{region '#Template'}
	{attribute 'Version' := '5.2.1.0'}
	{attribute 'Tags' := '"LCID": "1031", "Text": "RA, Sunprotection, Building"'}
	{attribute 'Tags' := '"LCID": "1033", "Text": "RA, Sunprotection, Building"'}
	{attribute 'Using' := '"Type": "Template", "URI": "Site"'}
	{attribute 'Using' := '"Type": "Template", "URI": "BA2_Param"'}
	{attribute 'Using' := '"Type": "Template", "URI": "EC_ID"'}
	{attribute 'Using' := '"Type": "Template", "URI": "ST_BA_BuildingSunblind"'}
	{attribute 'Using' := '"Type": "Template", "URI": "ST_BA_Sunblind"'}
	{attribute 'Using' := '"Type": "Template", "URI": "E_BA_SunBldPrio"'}
	{attribute 'Description' := '"LCID": "1031", "Text": "Sonnenschutz Gebäudedaten"'}
	{attribute 'Description' := '"LCID": "1033", "Text": "Sunprotection building data"'}
{endregion}
FUNCTION_BLOCK FB_BA_BuildingSunprotection EXTENDS FB_BA_View
VAR_INPUT CONSTANT	
	FireAlert					: FB_BA_SunBldEvt			:=(ePrio:=E_BA_SunBldPrio.eFire);	
	Burglary					: FB_BA_SunBldEvt			:=(ePrio:=E_BA_SunBldPrio.eBurglary);	
	IceProtection				: FB_BA_IceProtection;  
	GlobalThAutoRlse			: FB_BA_Hys_03;
	GlobalTwiLgtAutoRlse		: FB_BA_Hys_03;
	SunPrtcPosIntval			: FB_BA_AV_Op_SP;       
	GlobalResetManMode			: FB_BA_BV_Op_Val;   
END_VAR

VAR
	BuildingAlarms				: FB_BA_SunBldTgmSel4;	
	rtManResetEnergLvl			: R_TRIG;	
END_VAR
VAR // added by the converter: edge detectors and wires of the graphical bodies
    _s1 : ST_BA_BuildingSunblind;
    _w1 : UDINT;
END_VAR

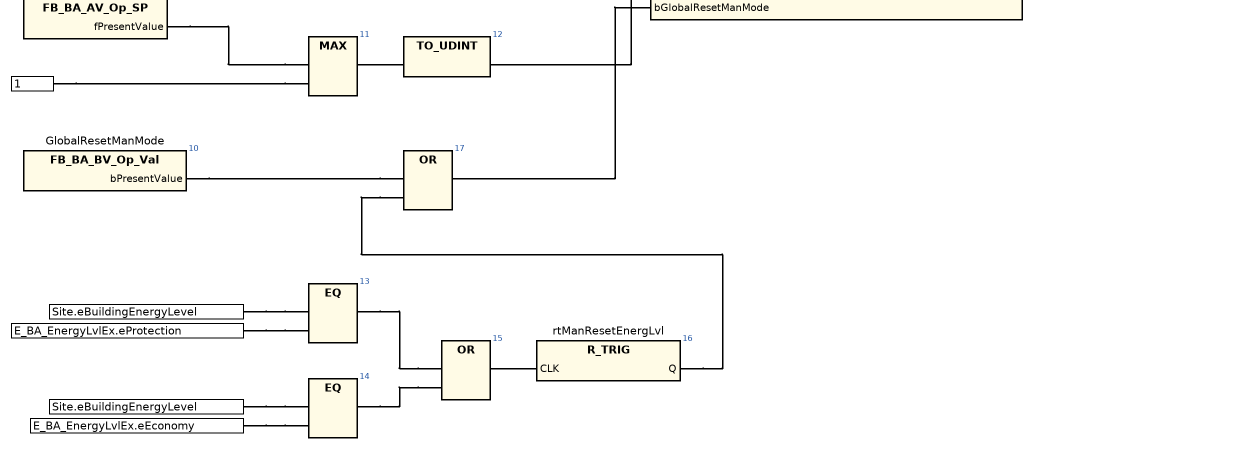
SUPER^(); // FB_BA_View
IceProtection(); // FB_BA_IceProtection
// ----------------------------------------  common alarms  ----------------------------------------
FireAlert(bEn := Site.stBuildingAlarms.bFireAlert, fPos := 0.0, fAngl := 0.0); // FB_BA_SunBldEvt
Burglary(bEn := Site.stBuildingAlarms.bBurglary, fPos := 0.0, fAngl := 0.0); // FB_BA_SunBldEvt
BuildingAlarms(
    stSunBldTgm_1 := FireAlert.stSunBld,
    stSunBldTgm_2 := Burglary.stSunBld,
    stSunBldTgm_3 := IceProtection.stSunBld); // FB_BA_SunBldTgmSel4
// ----------------------------------------  global criteria thermo- and twilight-automatic  ----------------------------------------
GlobalThAutoRlse(bEn := TRUE, fIn := Site.stWeatherStation.fGlobalRadiation); // FB_BA_Hys_03
GlobalTwiLgtAutoRlse(bEn := TRUE, fIn := (Site.stWeatherStation.fBrightnessNorth + Site.stWeatherStation.fBrightnessEast + Site.stWeatherStation.fBrightnessSouth + Site.stWeatherStation.fBrightnessWest) / 4); // FB_BA_Hys_03
// ----------------------------------------  assembling building-data-telegram  ----------------------------------------
SunPrtcPosIntval(); // FB_BA_AV_Op_SP
GlobalResetManMode(); // FB_BA_BV_Op_Val
_w1 := TO_UDINT(MAX(SunPrtcPosIntval.fPresentValue, 1));
rtManResetEnergLvl(CLK := Site.eBuildingEnergyLevel = E_BA_EnergyLvlEx.eProtection OR Site.eBuildingEnergyLevel = E_BA_EnergyLvlEx.eEconomy); // R_TRIG
// compose _s1 : ST_BA_BuildingSunblind
_s1.stSunBld := BuildingAlarms.stSunBld;
_s1.bGlobalThAuto_Release := GlobalThAutoRlse.bPresentValue;
_s1.bGlobalTwiLgtAuto_Release := GlobalTwiLgtAutoRlse.bPresentValue;
_s1.nSunPrtc_PositionInterval := _w1;
_s1.bGlobalResetManMode := GlobalResetManMode.bPresentValue OR rtManResetEnergLvl.Q;
Site.stBuildingSunBlind := _s1;

METHOD FB_init : BOOL
VAR_INPUT
	bInitRetains : BOOL; // if TRUE; the retain variables are initialized (warm start / cold start)
	bInCopyCode : BOOL;  // if TRUE; the instance afterwards gets moved into the copy code (online change)
END_VAR
IceProtection.iParent					:= THIS^;	
IceProtection.iLabel					:= LblCtl_IceProtection;
IceProtection.sObjectName		   		:= '{Idx=01}';
IceProtection.eDPADMode					:= E_BA_DPADMode.eInclude;
                                    	
GlobalThAutoRlse.iParent				:= THIS^;	
GlobalThAutoRlse.iLabel					:= LblCtl_ThermoAutomatic;
GlobalThAutoRlse.sObjectName			:= '{Idx=01}';
GlobalThAutoRlse.eDPADMode				:= E_BA_DPADMode.eInclude;
GlobalThAutoRlse.fOnMax					:= 10000;
GlobalThAutoRlse.fOffMax				:= 10000;
GlobalThAutoRlse.On.iLabel				:= LblCtl_RadiationOn;
GlobalThAutoRlse.On.sObjectName			:= '{Idx=01}';
GlobalThAutoRlse.On.eUnit				:= E_BA_Unit.eLight_WattsPerSquareMeter; 
GlobalThAutoRlse.On.fValueRm			:= 800.0;
GlobalThAutoRlse.Off.iLabel				:= LblCtl_RadiationOff;
GlobalThAutoRlse.Off.sObjectName		:= '{Idx=02}';
GlobalThAutoRlse.Off.eUnit				:= E_BA_Unit.eLight_WattsPerSquareMeter; 
GlobalThAutoRlse.Off.fValueRm			:= 200.0;
GlobalThAutoRlse.DlyOn.iLabel			:= LblCtl_RadiationDlyOn;
GlobalThAutoRlse.DlyOn.eUnit			:= E_BA_Unit.eTime_Seconds; 
GlobalThAutoRlse.DlyOn.fValueRm			:= 180.0;
GlobalThAutoRlse.DlyOff.iLabel			:= LblCtl_RadiationDlyOff;
GlobalThAutoRlse.DlyOff.eUnit			:= E_BA_Unit.eTime_Seconds;
GlobalThAutoRlse.DlyOff.fValueRm		:= 180.0;
GlobalThAutoRlse.Q.iLabel				:= LblCtl_GlobalThermoAutomaticRelease;
                                    	
GlobalTwiLgtAutoRlse.iParent			:= THIS^;	
GlobalTwiLgtAutoRlse.iLabel				:= LblCtl_TwilightAutomatic;
GlobalTwiLgtAutoRlse.sObjectName		:= '{Idx=01}';
GlobalTwiLgtAutoRlse.eDPADMode			:= E_BA_DPADMode.eInclude;
GlobalTwiLgtAutoRlse.fOnMax				:= 2000;
GlobalTwiLgtAutoRlse.fOffMax			:= 2000;
GlobalTwiLgtAutoRlse.On.iLabel			:= LblCtl_BrightnessOn;
GlobalTwiLgtAutoRlse.On.sObjectName		:= '{Idx=01}';
GlobalTwiLgtAutoRlse.On.eUnit			:= E_BA_Unit.eLight_Luxes; 
GlobalTwiLgtAutoRlse.On.fValueRm		:= 150.0;
GlobalTwiLgtAutoRlse.Off.iLabel			:= LblCtl_BrightnessOff;
GlobalTwiLgtAutoRlse.Off.sObjectName	:= '{Idx=02}';
GlobalTwiLgtAutoRlse.Off.eUnit			:= E_BA_Unit.eLight_Luxes; 
GlobalTwiLgtAutoRlse.Off.fValueRm		:= 200.0;
GlobalTwiLgtAutoRlse.DlyOn.iLabel		:= LblCtl_BrightnessDlyOn;
GlobalTwiLgtAutoRlse.DlyOn.eUnit		:= E_BA_Unit.eTime_Seconds; 
GlobalTwiLgtAutoRlse.DlyOn.fValueRm		:= 180.0;
GlobalTwiLgtAutoRlse.DlyOff.iLabel		:= LblCtl_BrightnessDlyOff;
GlobalTwiLgtAutoRlse.DlyOff.eUnit		:= E_BA_Unit.eTime_Seconds;
GlobalTwiLgtAutoRlse.DlyOff.fValueRm	:= 180.0;
GlobalTwiLgtAutoRlse.Q.iLabel			:= LblCtl_GlobalTwilightAutomaticRelease;
                              	    	
SunPrtcPosIntval.iParent				:= THIS^;
SunPrtcPosIntval.iLabel					:= LblCtl_SunProtectionInterval;	
SunPrtcPosIntval.eDPADMode				:= E_BA_DPADMode.eInclude;
SunPrtcPosIntval.SP.iLabel				:= LblFun_Setpoint;		
SunPrtcPosIntval.SP.eUnit				:= E_BA_Unit.eTime_Minutes; 
SunPrtcPosIntval.SP.fValueRm			:= 30;
SunPrtcPosIntval.SP.fCOVIncrement		:= BA2_Param.fDefCOVIncrement;		
                                    	
GlobalResetManMode.iParent				:= THIS^;	
GlobalResetManMode.iLabel				:= LblCtl_GlobalResetManMode;		
GlobalResetManMode.eDPADMode			:= E_BA_DPADMode.eInclude;
GlobalResetManMode.Val.iLabel			:= LblFun_Button;    
GlobalResetManMode.Val.sActiveText		:= txtEvent_On;  
GlobalResetManMode.Val.sInactiveText	:= txtEvent_Off;
GlobalResetManMode.Val.bValueRm			:= FALSE;  
GlobalResetManMode.Val.eToggleMode		:= E_BA_ToggleMode.ePushButton;
END_METHOD

END_FUNCTION_BLOCK

(* stored: Version 1.1.0.1, ProductVersion 3.1.4024.12
   POU FB_BA_BuildingSunprotection: Id {a80f4c80-c5dc-4d92-9550-21075fc22d4c}, SpecialFunc None
   Method FB_init: Id {1d9235ff-4925-4a07-88a7-371b84e07bf8} *)
